FUNCTION_BLOCK FB_AutoReset
// Automatically resets the boolean Value after the time period
VAR_INPUT
    Value : REFERENCE TO BOOL;
    PT : TIME;
END_VAR
VAR
    TON1 : TON;
END_VAR

TON1(IN := Value, PT := PT);
IF TON1.Q THEN
    Value := FALSE;
END_IF

END_FUNCTION_BLOCK

(* stored: Version 1.1.0.1, ProductVersion 3.1.4024.3
   POU FB_AutoReset: Id {2cb36d53-07de-4cd2-ab56-ddaa4f2bfa39}, SpecialFunc None *)
